// Mitsubishi GX Works2 project: check plc   PLC: FX3U/FX3UC

PROGRAM MAIN
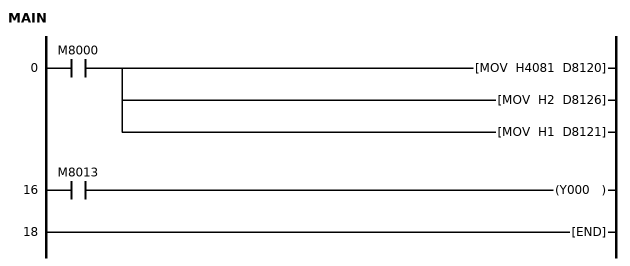
0     LD      M8000
      MOV     H4081 D8120
      MOV     H2 D8126
      MOV     H1 D8121
16    LD      M8013
      OUT     Y000
18    END
END_PROGRAM
